FUNCTION_BLOCK FB_HMIEMenu EXTENDS FB_BaseControlElement IMPLEMENTS ITF_HMIEMenu
VAR
	arrButtons		: ARRAY [0..GVL_HMIEConstans.MAX_NUMBER_OF_BUTTON_IN_MENU] OF ITF_HMIEButton;
	iNumerOfButton	: INT := -1;	//ilosć przycisków w menu
	
END_VAR

METHOD PUBLIC AddButton : BOOL
VAR_INPUT
	fbButton			: FB_HMIEButton;
END_VAR
IF (THIS^.iNumerOfButton + 1 <= GVL_HMIEConstans.MAX_NUMBER_OF_BUTTON_IN_MENU) THEN
	THIS^.iNumerOfButton := THIS^.iNumerOfButton + 1;
	THIS^.arrButtons [THIS^.iNumerOfButton] := fbButton;
	THIS^.arrButtons [THIS^.iNumerOfButton].SetEnable (bIN := TRUE);
	THIS^.arrButtons [THIS^.iNumerOfButton].SetVisible (bIN := TRUE);
	AddButton := TRUE;
ELSE
	AddButton := FALSE;
END_IF
END_METHOD

METHOD IsActiveButton : BOOL
VAR_INPUT
	iButton		: INT;	//numer przycisku
	bIN			: BOOL;
END_VAR
IsActiveButton	:= THIS^.arrButtons [iButton].IsActive ();
END_METHOD

METHOD IsEnableButton : BOOL
VAR_INPUT
	iButton		: INT;	//numer przycisku
	bIN			: BOOL;
END_VAR
IsEnableButton	:= THIS^.arrButtons [iButton].IsEnable ();
END_METHOD

METHOD IsVisibleButton : BOOL
VAR_INPUT
	iButton		: INT;	//numer przycisku
	bIN			: BOOL;
END_VAR
IsVisibleButton	:= THIS^.arrButtons [iButton].IsVisible ();
END_METHOD

METHOD SetActiveButton : BOOL
VAR_INPUT
	iButton		: INT;	//numer przycisku
	bIN			: BOOL;
END_VAR
THIS^.arrButtons [iButton].SetActive (bIN := bIN);
END_METHOD

METHOD SetEnableButton : BOOL
VAR_INPUT
	iButton		: INT;	//numer przycisku
	bIN			: BOOL;
END_VAR
THIS^.arrButtons [iButton].SetEnable (bIN := bIN);
END_METHOD

METHOD SetVisibleButton : BOOL
VAR_INPUT
	iButton		: INT;	//numer przycisku
	bIN			: BOOL;
END_VAR
THIS^.arrButtons [iButton].SetVisible (bIN := bIN);
END_METHOD

END_FUNCTION_BLOCK

(* stored: Version 1.1.0.1
   POU FB_HMIEMenu: Id {aca5b8d6-8bd3-4247-801c-4d7202167bd3}, SpecialFunc None
   Folder ITF_HMIEMenu: Id {4b3a4679-e153-0f1c-0cf6-c4b1dfee1813}
   Method AddButton: Id {84c5fa09-21a3-408e-a468-e17b66190995}
   Method IsActiveButton: Id {b4d1a0ff-bd9d-0a66-1dc5-0550ed0d188d}
   Method IsEnableButton: Id {217e2c6a-563a-08bd-0fa4-1cc88765e86d}
   Method IsVisibleButton: Id {20df5edd-f349-000a-1620-91b9a13457e8}
   Method SetActiveButton: Id {4a3f2cd9-b9dc-0e5a-20ae-b9e5849184e6}
   Method SetEnableButton: Id {09238708-59e8-0f4e-3df3-b9bd70508c9d}
   Method SetVisibleButton: Id {9b32dc56-5171-0eb1-09b1-fe51305e187e} *)
